(* CoDeSys 2.3.9.28 project: test.pro *)
(* Libraries: SysLibTime.lib 2.12.10 13:48:32, Standard.lib 2.12.10 13:48:34, SYSLIBCALLBACK.LIB 2.12.10 13:48:32 *)

(* PLC configuration (modules and I/O channels)
K-Bus [K_Bus] node 0, in %IB0 out %QB0
Fieldbus variables [FB_VARS] node 1, in %IB0 out %QB0
Flag variables [FLAG_VARS] node 2, in %IB0 out %QB0
*)

(* POU PLC_PRG, CFC *)
PROGRAM PLC_PRG
VAR
	a: IntervalSepnuti;
	x: BOOL;
	cas_datum: CurTimeEx;
	System_cas: SysTime64;
	System_datum: SystemTimeDate;
	t: INT;
	z: INT;
END_VAR
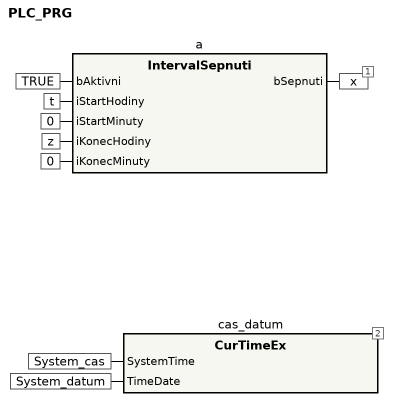
_CFC_ (* Continuous Function Chart, elements in execution order *)
#0 a:IntervalSepnuti(bAktivni: TRUE, iStartHodiny: t, iStartMinuty: 0, iKonecHodiny: z, iKonecMinuty: 0)
#1 x <= #0.bSepnuti
#2 cas_datum:CurTimeEx(SystemTime: System_cas, TimeDate: System_datum)
_END_CFC_
(* the same logic as Structured Text *)
a(bAktivni := TRUE, iStartHodiny := t, iStartMinuty := 0, iKonecHodiny := z, iKonecMinuty := 0);
x := a.bSepnuti;
cas_datum(SystemTime := System_cas, TimeDate := System_datum);
END_PROGRAM

(* POU Ostatni/IntervalSepnuti, ST *)
FUNCTION_BLOCK IntervalSepnuti
VAR_INPUT
	bAktivni: BOOL;
	iStartHodiny: INT;
	iStartMinuty: INT;
	iKonecHodiny: INT;
	iKonecMinuty: INT;
END_VAR
VAR_OUTPUT
	bSepnuti: BOOL;
END_VAR
VAR
END_VAR
IF (bAktivni)
THEN
	IF(iStartHodiny = 12 )
	THEN
		IF(iStartMinuty <= 35)
		THEN
			bSepnuti:= TRUE;
		END_IF
	ELSIF (iStartHodiny < 12)
	THEN
		bSepnuti := TRUE;
	ELSE
		bSepnuti := FALSE;
	END_IF

	IF(iKonecHodiny = 12)
	THEN
		IF(iKonecMinuty <= 35)
		THEN
			bSepnuti := FALSE;
		END_IF

	ELSIF(iKonecHodiny < 12)
	THEN
		bSepnuti := FALSE;
	ELSE
		bSepnuti := TRUE;
	END_IF
END_IF
END_FUNCTION_BLOCK
